// TIA Portal V17 export
// export: Created 2021-12-03T08:12:56.3832063Z, ExportSetting WithDefaults, DisplayName Totally Integrated Automation Portal, DisplayVersion V17, DisplayName TIA Portal Openness, DisplayVersion V17, DisplayName TIA Portal Version Control Interface, DisplayVersion V17, DisplayName STEP 7 Professional, DisplayVersion V17, DisplayName STEP 7 Safety, DisplayVersion V17, DisplayName WinCC Advanced, DisplayVersion V17
FUNCTION_BLOCK "FB_GnrlFunc"   // FB30, FBD
VERSION : 0.1
// stored: AutoNumber false, IsIECCheckEnabled false, UDAEnableTagReadback false
   VAR DB_SPECIFIC
      AxSR : Struct
         SrvcMd : Bool;
      END_STRUCT;
   END_VAR
BEGIN

REGION Network 1: Сервисный режим
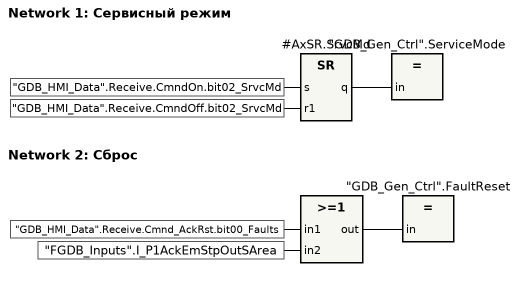
   IF "GDB_HMI_Data".Receive.CmndOn.bit02_SrvcMd THEN
       #AxSR.SrvcMd := TRUE;   // SR flip-flop
   END_IF;
   IF "GDB_HMI_Data".Receive.CmndOff.bit02_SrvcMd THEN #AxSR.SrvcMd := FALSE; END_IF;
   "GDB_Gen_Ctrl".ServiceMode := #AxSR.SrvcMd;
END_REGION

REGION Network 2: Сброс
   "GDB_Gen_Ctrl".FaultReset := "GDB_HMI_Data".Receive.Cmnd_AckRst.bit00_Faults OR "FGDB_Inputs".I_P1AckEmStpOutSArea;
END_REGION
END_FUNCTION_BLOCK
